{attribute 'GeneratedUsingTerminal: '}
{attribute addProperty BoxType ""}
{attribute addProperty Id "unreferencedAT %I*SyncUnitTask_AB2F50799PlcTaskAT %I*SyncUnitTask_AB2F50799"}
{attribute addProperty CRC "1272976489"}
{attribute addProperty Size "18"}
TYPE SyncUnitTasks_4BE01469 EXTENDS TcoIo.SyncUnitTasksBase_7C8711EB :
STRUCT
	{attribute addProperty Name "unreferenced"}
	unreferenced : TcoIo.SyncUnitTask_AB2F5079;
	{attribute addProperty Name "PlcTask"}
	PlcTask : TcoIo.SyncUnitTask_AB2F5079;
END_STRUCT
END_TYPE

(* stored: Version 1.2.0.0
   DUT SyncUnitTasks_4BE01469: Id {2feeeae3-7b11-4455-94e6-f73efdf05bb5} *)
